TYPE ST_ThNTZ_Aktor :
STRUCT
	Verfuegbarkeit_Heizer		: BOOL;
	Verfuegbarkeit_Kuehler	: BOOL;
	Betrieb_Heizer_Anford		: BOOL;
	Betrieb_Kuehler_Anford	: BOOL;
END_STRUCT
END_TYPE

(* stored: Version 1.1.0.1, ProductVersion 3.1.4024.9
   DUT ST_ThNTZ_Aktor: Id {16ae6afd-cd7c-4218-ab19-2f68efa74a9c} *)
